// TIA Portal V19 export
VAR_GLOBAL   // PLC tag table "Default tag table"
   Tag_111 AT %MW1 : Int;
   di_1 AT %I0.0 : Bool;
   di_2 AT %I0.1 : Bool;
   ai_raw_01 AT %IW272 : Int;
   ai_raw_02 AT %IW274 : Int;
   ai_raw_03 AT %IW276 : Int;
   ai_raw_04 AT %IW278 : Int;
END_VAR
VAR_GLOBAL CONSTANT   // user constants
   C_HW_MAX : Int := 27648;
   C_HW_MIN : Int := 0;
   C_DIAG_OVER : Real := 1.1759;
   C_DIAG_UNDER : Real := -0.1759;
END_VAR
